// TIA Portal V20 export
TYPE "LConSMC_typeTorquePrecontrolDiag"
// Diagnose der Drehmomentenvorsteuerung / Diagnostic structure for torque precontrol
// stored: Access Published
   STRUCT
      upperTorqueLimit : LReal := 0.0;   // [Einheit der Achse] Obere Drehmomentengrenze / [Unit of the axis] Upper torque limit
      lowerTorqueLimit : LReal := 0.0;   // [Einheit der Achse] Untere Drehmomentengrenze / [Unit of the axis] Lower torque limit
      totalTorquePreControl : LReal := 0.0;   // [Einheit der Achse] Gesamtes Vorsteuerdrehmoment / [Unit of the axis] Total torque precontrol value
      totalInertia : LReal;   // [kgm^2 oder lbft^2] Aktuelle Trägheit des Wicklers / [kgm^2 or lbft^2] Current intertia of the winder
      maxInertia : LReal;   // [kgm^2 or lbft^2] Maximale Trägheit bei maximalem Durchmesser / [kgm^2 or lbft^2] Maximum inertia at maximum diameter
      referenceTorque : LReal;   // Verwendetes Referenzdrehmoment / Used reference torque value
      loadGear { S7_SetPoint := 'True'} : "LConSMC_typeLoadGear";   // Ausgelesene Getriebeübersetzung / Gear ratio read out
   END_STRUCT;
END_TYPE
